# B&R Automation Studio project wtf_is_this
Automation Studio 4.5.2.102; technology packages: Acp10Arnc0 5.2.1

## Configuration Config1

### Task classes (Cpu.sw)
```
Cyclic#1 (cycle 2000 us, tolerance 0 us):
  ncsdcctrl <- ncsdcctrl.prg
Cyclic#8:
  Program <- Program.prg
  Program1 <- Program1.prg
DataObjects: Acp10sys
NcDataObjects: acp10etxen <- acp10etxen.dob, gAxis01a <- gAxis01obj.gAxis01a.dob, gAxis01i <- gAxis01obj.gAxis01i.dob
VcDataObjects: Visu <- Visu.dob
Binaries: udbdef, TCData, vcpdsw, vcrt, vcpfmtcx, vccslider, Visu03, vcfile, vcgclass, arial, vccbmp, vcmgr, vcchspot, vcdsloc, vcfntttf, Visu02, vccovl, vcshared, arialbd, vcalarm, vcptelo, vcpdpp30, Visu01, vcbclass, vcpfpp30, vcdsint, vctcal, vcctext, vccbtn, ashwac, arconfig, asfw, User, ashwd, iomap, Role, sysconf, acp10cfg, Acp10map, arsvcreg
Libraries: Library, Acp10par, NcGlobal, Acp10man, Acp10sdc, Acp10_MC, brsystem, sys_lib, runtime, AsBrStr, vcresman, asieccon, fileio, astime, dataobj, powerlnk
```

### Hardware
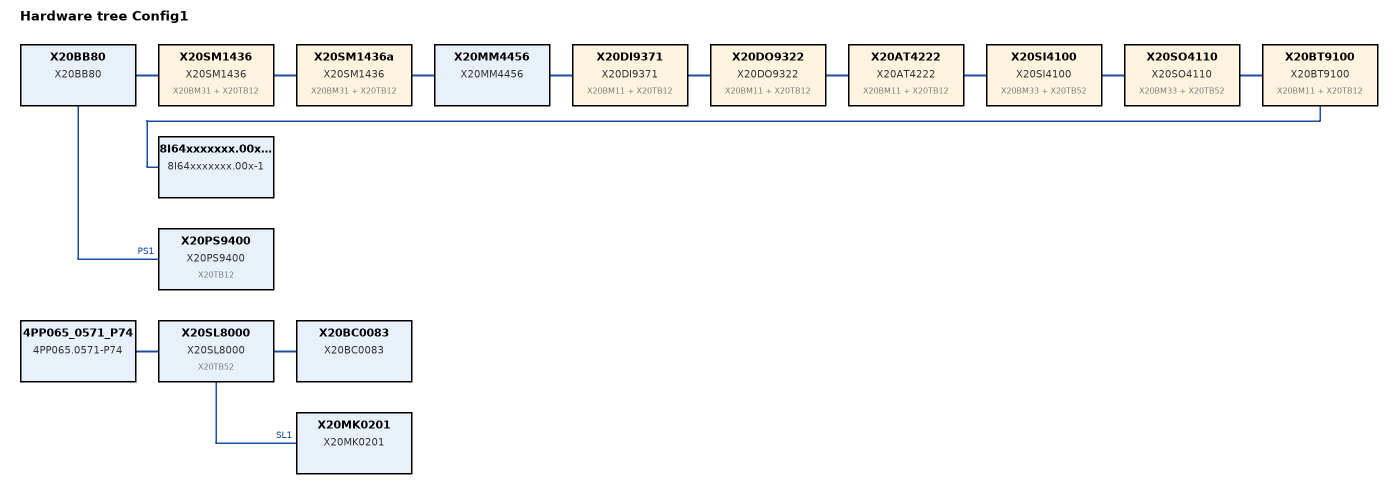
```
4PP065_0571_P74 : 4PP065.0571-P74 v1.1.2.0
  Connector IF5:
    ActivateDevice = 1
    Mode = Manual
    InternetAddress = 10.0.1.10
    Vnc1
    VncVcObjectName1 = Visu
    VncKeyMappingFile1 = VC\PS2-Keyboard.dis
  ConfigurationID = 1234_Config1
  TimerDeviceType = EPLX2X
  TimerDevice = 4PP065_0571_P74.IF4
  TaskClassIdleTime = 2000
  Cyclic1Duration = 2000
  Cyclic1Tolerance = 0
  Cyclic1Output = 1
  VcObjectName = Visu
8I64xxxxxxx.00x-1 : 8I64xxxxxxx.00x-1 v2.1.3.0  [X2X1 -> X20BT9100.X2X1 [Cable Type=X2XCable, Length=10, Version=1.0.0.2]]
  packedETAD = packed
  packedCMDD = packed
X20AT4222 : X20AT4222 v1.2.3.0  [SS1 -> X20TB12e.SS; SL -> X20BM11b.SL1]
X20BB80 : X20BB80 v1.0.2.0
X20BC0083 : X20BC0083 v2.14.0.0  [PLK1 -> X20SL8000.PLK2 [Cable Type=PowerlinkCable, Length=10, Version=1.0.0.2]; SL -> X20BB80.SL1]
X20BM11 : X20BM11 v1.0.0.1  [X2X1 -> X20MM4456.X2X2]
X20BM11a : X20BM11 v1.0.0.1  [X2X1 -> X20BM11.X2X2]
X20BM11b : X20BM11 v1.0.0.1  [X2X1 -> X20BM11a.X2X2]
X20BM11c : X20BM11 v1.0.0.1  [X2X1 -> X20BM33a.X2X2]
X20BM31 : X20BM31 v1.0.0.1  [X2X1 -> X20BB80.IF1]
X20BM31a : X20BM31 v1.0.0.1  [X2X1 -> X20BM31.X2X2]
X20BM33 : X20BM33 v1.0.0.4 (Disabled=true)  [X2X1 -> X20BM11b.X2X2]
X20BM33a : X20BM33 v1.0.0.4 (Disabled=true)  [X2X1 -> X20BM33.X2X2]
X20BT9100 : X20BT9100 v1.0.3.0  [SS1 -> X20TB12f.SS; SL -> X20BM11c.SL1]
X20DI9371 : X20DI9371 v1.0.2.0  [SS1 -> X20TB12c.SS; SL -> X20BM11.SL1]
X20DO9322 : X20DO9322 v1.0.3.0  [SS1 -> X20TB12d.SS; SL -> X20BM11a.SL1]
X20MK0201 : X20MK0201 v1.0.0.0 (Disabled=true)  [SL -> X20SL8000.SL1]
X20MM4456 : X20MM4456 v1.4.0.0  [X2X1 -> X20BM31a.X2X2]
X20PS9400 : X20PS9400 v1.8.0.0  [SS1 -> X20TB12.SS; PS -> X20BB80.PS1]
X20SI4100 : X20SI4100 v1.10.1.1 (Disabled=true)  [SS1 -> X20TB52a.SS; SL -> X20BM33.SL1]
X20SL8000 : X20SL8000 v1.6.5.2 (Disabled=true)  [PLK1 -> 4PP065_0571_P74.IF4 [Cable Type=PowerlinkCable, Length=10, Version=1.0.0.2]; PLK2 -> X20BC0083.PLK1 [Cable Type=PowerlinkCable, Length=10, Version=1.0.0.2]; SS1 -> X20TB52.SS]
  SafeProject = SafeLOGIC-1
X20SM1436 : X20SM1436 v2.3.0.0  [SS1 -> X20TB12a.SS; SL -> X20BM31.SL1]
X20SM1436a : X20SM1436 v2.3.0.0  [SS1 -> X20TB12b.SS; SL -> X20BM31a.SL1]
X20SO4110 : X20SO4110 v1.10.12.0 (Disabled=true)  [SS1 -> X20TB52b.SS; SL -> X20BM33a.SL1]
  SafeModuleID = 3
X20TB12 : X20TB12 v1.0.0.0
X20TB12a : X20TB12 v1.0.0.0
X20TB12b : X20TB12 v1.0.0.0
X20TB12c : X20TB12 v1.0.0.0
X20TB12d : X20TB12 v1.0.0.0
X20TB12e : X20TB12 v1.0.0.0
X20TB12f : X20TB12 v1.0.0.0
X20TB52 : X20TB52 v1.0.0.1 (Disabled=true)
X20TB52a : X20TB52 v1.0.0.1 (Disabled=true)
X20TB52b : X20TB52 v1.0.0.1 (Disabled=true)
```

### IoMap.iom - 4PP065_0571_P74/IoMap.iom
```iecst
VAR_CONFIG
	::Program:lamps[0] AT %QX."X20DO9322".DigitalOutput02;
	::Program:lamps[1] AT %QX."X20DO9322".DigitalOutput03;
	::Program:lamps[2] AT %QX."X20DO9322".DigitalOutput04;
	::Program:lamps[3] AT %QX."X20DO9322".DigitalOutput05;
	::Program:lamp_speed AT %IX."X20DI9371".DigitalInput01;
	::Program1:state.STATE AT %IW."8I64xxxxxxx.00x-1".ETAD_Input;
	::Program1:state.COM AT %QW."8I64xxxxxxx.00x-1".CMDD_Output;
	::Program1:target_speed AT %QW."8I64xxxxxxx.00x-1".LFRD_Output;
	Cyclic#1.gAxis01_DrvIf.iLifeCnt AT %IB."8I64xxxxxxx.00x-1".SDC_LifeCnt;
	Cyclic#1.gAxis01_DrvIf.iDrvOK AT %IX."8I64xxxxxxx.00x-1".ETAD_Input_Bool_02;
	Cyclic#1.gAxis01_DrvIf.oSetTime AT %QW."8I64xxxxxxx.00x-1".SDC_SetTime;
	Cyclic#1.gAxis01_DiDoIf.iLifeCntDriveReady AT %IB."8I64xxxxxxx.00x-1".SDC_LifeCnt;
	Cyclic#1.gAxis01_DiDoIf.iLifeCntDriveEnable AT %IB."8I64xxxxxxx.00x-1".SDC_LifeCnt;
	Cyclic#1.gAxis01_DiDoIf.oDriveEnable AT %QX."8I64xxxxxxx.00x-1".CMDD_Output_Bool_00;
	Cyclic#1.gAxis01_ModuleOk AT %QX."8I64xxxxxxx.00x-1".CMDD_Output_Bool_01;
	Cyclic#1.gAxis01_ModuleOk AT %QX."8I64xxxxxxx.00x-1".CMDD_Output_Bool_02;
	Cyclic#1.gAxis01_ModuleOk AT %IX."8I64xxxxxxx.00x-1".ModuleOk;
	Cyclic#1.gAxis01_DiDoIf.oDriveEnable AT %QX."8I64xxxxxxx.00x-1".CMDD_Output_Bool_03;
	Cyclic#1.gAxis01_DiDoIf.iDriveReady AT %IX."8I64xxxxxxx.00x-1".ETAD_Input_Bool_02;
	::Program1:RFRD_Input AT %IW."8I64xxxxxxx.00x-1".RFRD_Input;
END_VAR
```

## Logical view

Binary libraries used (declarations not repeated): operator, runtime, astime, AsIecCon, Acp10par, NcGlobal, Acp10man, Acp10sdc, Acp10_MC, brsystem, sys_lib, AsBrStr

### Global.var - Global variables
```iecst
VAR
	gAxis01 : ACP10AXIS_typ;
	gAxis01_HW : SdcHwCfg_typ := (0);
	gAxis01_DrvIf : SdcDrvIf16_typ := (0);
	gAxis01_DiDoIf : SdcDiDoIf_typ := (0);
	gAxis01_ModuleOk : BOOL := 0;
END_VAR
```


### Program Logical/Program (ANSIC)

#### Variables.var
```iecst
VAR
	lamps : ARRAY[0..3] OF BOOL;
	button_colors : ARRAY[0..3] OF UINT;
	lamp_speed : BOOL;
	enabled : BOOL;
END_VAR
```

#### Main.c
```c
#include <bur/plctypes.h>

#ifdef _DEFAULT_INCLUDES
	#include <AsDefault.h>
#endif

int current = 0;
UDINT time = 0;

void _INIT ProgramInit(void)
{

}

void _CYCLIC ProgramCyclic(void)
{
	if (enabled == 1) {
		if (time >= (lamp_speed ? 20 : 30)) {
			lamps[current] = 0;
			current = (current + 1) % 4;
			lamps[current] = 1;

			time = 0;
		}
	}
	++time;
}

void _EXIT ProgramExit(void)
{

}
```

- Visualisation Logical/Visu (not shown)

### Library Logical/Library (ANSIC)

#### Constants.var - Exported constants
```iecst
VAR CONSTANT
	CMD_SWITCHED_ON : USINT := 7;
	CMD_ENABLED : USINT := 15;
	CMD_SHUTDOWN : USINT := 6;
	STATE_READY : USINT := 33;
	STATE_DISABLED : USINT := 64;
	STATE_SWITCHED_ON : USINT := 35;
END_VAR
```

#### Library.fun - Exported functions and function blocks
```iecst
{REDUND_ERROR} FUNCTION_BLOCK state_machine (*TODO: Add your comment here*) (*$GROUP=User,$CAT=User,$GROUPICON=User.png,$CATICON=User.png*)
	VAR_INPUT
		ENABLE : BOOL;
		STATE : UINT;
	END_VAR
	VAR_OUTPUT
		COM : UINT;
	END_VAR
END_FUNCTION_BLOCK
```

#### State.c
```c
#include <bur/plctypes.h>
#ifdef __cplusplus
	extern "C"
	{
#endif
	#include "Library.h"
#ifdef __cplusplus
	};
#endif

UINT get_cmd(UINT cur_state) {
	switch (cur_state) {
		case STATE_DISABLED:
			return CMD_SHUTDOWN;
		case STATE_READY:
			return CMD_ENABLED;
		case STATE_SWITCHED_ON:
			return CMD_SWITCHED_ON;
	}
}

void state_machine(struct state_machine* inst) {
	if (!inst->ENABLE) {
		inst->COM = CMD_SHUTDOWN;
	} else {
		UINT new_cmd = get_cmd(inst->STATE & 0x6f);
		inst->COM = new_cmd;
	}
}
```

### Program Logical/Program1 (ANSIC)

#### Variables.var
```iecst
VAR
	target_speed : INT := 0;
	real_speed : INT;
	state : state_machine;
	RFRD_Input : INT;
END_VAR
```

#### Main.c
```c
#include <bur/plctypes.h>

#ifdef _DEFAULT_INCLUDES
	#include <AsDefault.h>
#endif

void _INIT ProgramInit(void)
{
	target_speed = 500;
	state.ENABLE = 1;
}

void _CYCLIC ProgramCyclic(void)
{
	real_speed = -RFRD_Input;

	state_machine(&state);
}

void _EXIT ProgramExit(void)
{

}
```

Listed in the project but not available here: Logical/Global.typ, Logical/Library/Types.typ, Logical/ncsdcctrl, Logical/acp10etxen, Logical/gAxis01obj
